{attribute 'qualified_only'}
{attribute 'strict'}
TYPE EResult_t :
(
	eStatePassed,
	eStateFailed,
	eStateFailedFatal
);
END_TYPE

(* stored: Version 1.1.0.1, ProductVersion 3.1.4022.9
   DUT EResult_t: Id {ab665a68-6565-4f52-bb64-6093dc936587} *)
